TEXTLIST tlTableBottlePlaceState
  0 = 'Empty'
  1 = 'BeforeWeighing'
  2 = 'Processing'
  3 = 'AfterWeighing'
  4 = 'NOK'
   = ''
END_TEXTLIST

(* stored: Version 1.1.0.1, ProductVersion 3.1.4024.15
   TextList tlTableBottlePlaceState: Id {719518ed-018f-4684-b3c6-d2b2c512f53b} *)
